TYPE DegreesMinutesSeconds :
STRUCT
    positive : BOOL;
    
    degrees : DINT;
    minutes : DINT;
    seconds : LREAL;
END_STRUCT
END_TYPE

(* stored: Version 1.1.0.1, ProductVersion 3.1.4018.5
   DUT DegreesMinutesSeconds: Id {56dffeaa-e654-4664-b98f-adf436dd344f} *)
